// TIA Portal V20 program export: 0 tag tables, 0 data types, 0 data blocks, 2 code blocks (in call order from the OBs), 0 instance data blocks

ORGANIZATION_BLOCK "Main"   // OB1, LAD, ProgramCycle
// stored: AutoNumber false
BEGIN

REGION Network 1
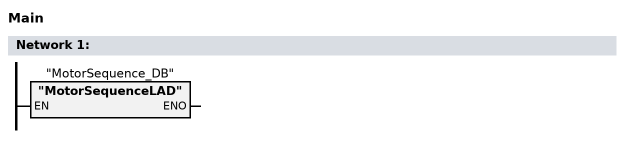
   RUNG wire#powerrail
      "MotorSequence_DB"()
   END_RUNG
   // the same network as SCL:
   "MotorSequence_DB"();   // "MotorSequenceLAD"
END_REGION
END_ORGANIZATION_BLOCK

FUNCTION_BLOCK "MotorSequenceLAD"   // FB1, LAD
{ S7_Optimized_Access := 'TRUE' }
// stored: AutoNumber true
   VAR
      Start2 { S7_SetPoint := 'True'} : TON_TIME;
      Start3 { S7_SetPoint := 'True'} : TON_TIME;
      Stop2 { S7_SetPoint := 'True'} : TON_TIME;
      Stop1 { S7_SetPoint := 'True'} : TON_TIME;
   END_VAR
BEGIN

REGION Network 1: 启动上升沿，仅接受新的按钮动作
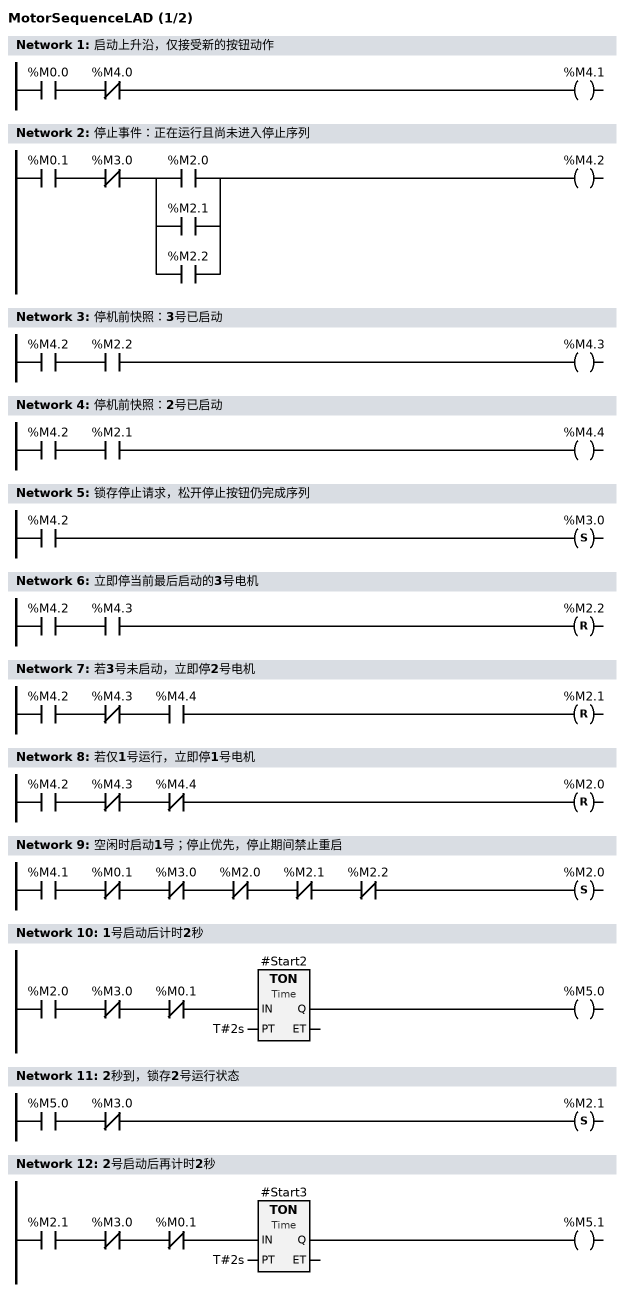
   RUNG wire#powerrail
      Contact( %M0.0 )
      I_Contact( %M4.0 )
      Coil( %M4.1 )
   END_RUNG
   // the same network as SCL:
   %M4.1 := %M0.0 AND NOT %M4.0;
END_REGION

REGION Network 2: 停止事件：正在运行且尚未进入停止序列
   %M4.2 := %M0.1 AND NOT %M3.0 AND (%M2.0 OR %M2.1 OR %M2.2);
END_REGION

REGION Network 3: 停机前快照：3号已启动
   RUNG wire#powerrail
      Contact( %M4.2 )
      Contact( %M2.2 )
      Coil( %M4.3 )
   END_RUNG
   // the same network as SCL:
   %M4.3 := %M4.2 AND %M2.2;
END_REGION

REGION Network 4: 停机前快照：2号已启动
   RUNG wire#powerrail
      Contact( %M4.2 )
      Contact( %M2.1 )
      Coil( %M4.4 )
   END_RUNG
   // the same network as SCL:
   %M4.4 := %M4.2 AND %M2.1;
END_REGION

REGION Network 5: 锁存停止请求，松开停止按钮仍完成序列
   RUNG wire#powerrail
      Contact( %M4.2 )
      S_Coil( %M3.0 )
   END_RUNG
   // the same network as SCL:
   IF %M4.2 THEN %M3.0 := TRUE; END_IF;
END_REGION

REGION Network 6: 立即停当前最后启动的3号电机
   RUNG wire#powerrail
      Contact( %M4.2 )
      Contact( %M4.3 )
      R_Coil( %M2.2 )
   END_RUNG
   // the same network as SCL:
   IF %M4.2 AND %M4.3 THEN %M2.2 := FALSE; END_IF;
END_REGION

REGION Network 7: 若3号未启动，立即停2号电机
   RUNG wire#powerrail
      Contact( %M4.2 )
      I_Contact( %M4.3 )
      Contact( %M4.4 )
      R_Coil( %M2.1 )
   END_RUNG
   // the same network as SCL:
   IF %M4.2 AND NOT %M4.3 AND %M4.4 THEN %M2.1 := FALSE; END_IF;
END_REGION

REGION Network 8: 若仅1号运行，立即停1号电机
   RUNG wire#powerrail
      Contact( %M4.2 )
      I_Contact( %M4.3 )
      I_Contact( %M4.4 )
      R_Coil( %M2.0 )
   END_RUNG
   // the same network as SCL:
   IF %M4.2 AND NOT %M4.3 AND NOT %M4.4 THEN %M2.0 := FALSE; END_IF;
END_REGION

REGION Network 9: 空闲时启动1号；停止优先，停止期间禁止重启
   RUNG wire#powerrail
      Contact( %M4.1 )
      I_Contact( %M0.1 )
      I_Contact( %M3.0 )
      I_Contact( %M2.0 )
      I_Contact( %M2.1 )
      I_Contact( %M2.2 )
      S_Coil( %M2.0 )
   END_RUNG
   // the same network as SCL:
   IF %M4.1 AND NOT %M0.1 AND NOT %M3.0 AND NOT %M2.0 AND NOT %M2.1 AND NOT %M2.2 THEN %M2.0 := TRUE; END_IF;
END_REGION

REGION Network 10: 1号启动后计时2秒
   RUNG wire#powerrail
      Contact( %M2.0 )
      I_Contact( %M3.0 )
      I_Contact( %M0.1 )
      { S7_Templates := "time_type := Time" } #Start2.TON(pt := T#2s, et =>)
      Coil( %M5.0 )
   END_RUNG
   // the same network as SCL:
   #Start2(IN := %M2.0 AND NOT %M3.0 AND NOT %M0.1, PT := T#2s);   // TON
   %M5.0 := #Start2.Q;
END_REGION

REGION Network 11: 2秒到，锁存2号运行状态
   RUNG wire#powerrail
      Contact( %M5.0 )
      I_Contact( %M3.0 )
      S_Coil( %M2.1 )
   END_RUNG
   // the same network as SCL:
   IF %M5.0 AND NOT %M3.0 THEN %M2.1 := TRUE; END_IF;
END_REGION

REGION Network 12: 2号启动后再计时2秒
   RUNG wire#powerrail
      Contact( %M2.1 )
      I_Contact( %M3.0 )
      I_Contact( %M0.1 )
      { S7_Templates := "time_type := Time" } #Start3.TON(pt := T#2s, et =>)
      Coil( %M5.1 )
   END_RUNG
   // the same network as SCL:
   #Start3(IN := %M2.1 AND NOT %M3.0 AND NOT %M0.1, PT := T#2s);   // TON
   %M5.1 := #Start3.Q;
END_REGION

REGION Network 13: 再过2秒，锁存3号运行状态
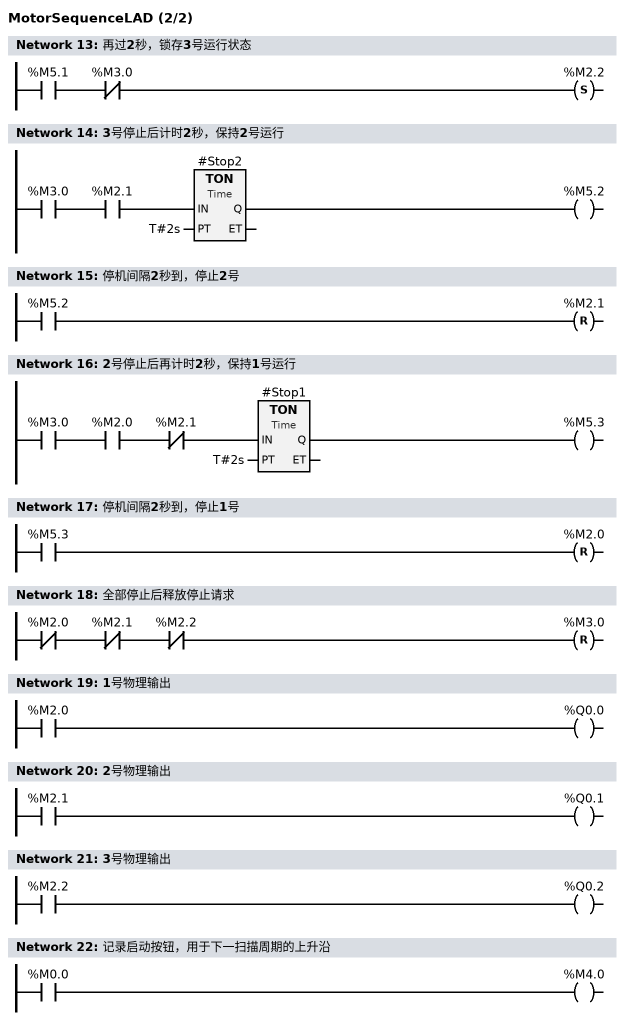
   RUNG wire#powerrail
      Contact( %M5.1 )
      I_Contact( %M3.0 )
      S_Coil( %M2.2 )
   END_RUNG
   // the same network as SCL:
   IF %M5.1 AND NOT %M3.0 THEN %M2.2 := TRUE; END_IF;
END_REGION

REGION Network 14: 3号停止后计时2秒，保持2号运行
   RUNG wire#powerrail
      Contact( %M3.0 )
      Contact( %M2.1 )
      { S7_Templates := "time_type := Time" } #Stop2.TON(pt := T#2s, et =>)
      Coil( %M5.2 )
   END_RUNG
   // the same network as SCL:
   #Stop2(IN := %M3.0 AND %M2.1, PT := T#2s);   // TON
   %M5.2 := #Stop2.Q;
END_REGION

REGION Network 15: 停机间隔2秒到，停止2号
   RUNG wire#powerrail
      Contact( %M5.2 )
      R_Coil( %M2.1 )
   END_RUNG
   // the same network as SCL:
   IF %M5.2 THEN %M2.1 := FALSE; END_IF;
END_REGION

REGION Network 16: 2号停止后再计时2秒，保持1号运行
   RUNG wire#powerrail
      Contact( %M3.0 )
      Contact( %M2.0 )
      I_Contact( %M2.1 )
      { S7_Templates := "time_type := Time" } #Stop1.TON(pt := T#2s, et =>)
      Coil( %M5.3 )
   END_RUNG
   // the same network as SCL:
   #Stop1(IN := %M3.0 AND %M2.0 AND NOT %M2.1, PT := T#2s);   // TON
   %M5.3 := #Stop1.Q;
END_REGION

REGION Network 17: 停机间隔2秒到，停止1号
   RUNG wire#powerrail
      Contact( %M5.3 )
      R_Coil( %M2.0 )
   END_RUNG
   // the same network as SCL:
   IF %M5.3 THEN %M2.0 := FALSE; END_IF;
END_REGION

REGION Network 18: 全部停止后释放停止请求
   RUNG wire#powerrail
      I_Contact( %M2.0 )
      I_Contact( %M2.1 )
      I_Contact( %M2.2 )
      R_Coil( %M3.0 )
   END_RUNG
   // the same network as SCL:
   IF NOT %M2.0 AND NOT %M2.1 AND NOT %M2.2 THEN %M3.0 := FALSE; END_IF;
END_REGION

REGION Network 19: 1号物理输出
   RUNG wire#powerrail
      Contact( %M2.0 )
      Coil( %Q0.0 )
   END_RUNG
   // the same network as SCL:
   %Q0.0 := %M2.0;
END_REGION

REGION Network 20: 2号物理输出
   RUNG wire#powerrail
      Contact( %M2.1 )
      Coil( %Q0.1 )
   END_RUNG
   // the same network as SCL:
   %Q0.1 := %M2.1;
END_REGION

REGION Network 21: 3号物理输出
   RUNG wire#powerrail
      Contact( %M2.2 )
      Coil( %Q0.2 )
   END_RUNG
   // the same network as SCL:
   %Q0.2 := %M2.2;
END_REGION

REGION Network 22: 记录启动按钮，用于下一扫描周期的上升沿
   RUNG wire#powerrail
      Contact( %M0.0 )
      Coil( %M4.0 )
   END_RUNG
   // the same network as SCL:
   %M4.0 := %M0.0;
END_REGION
END_FUNCTION_BLOCK
